// TIA Portal V19 export
FUNCTION_BLOCK "Decoiler_DiameterSensor_FB"   // FB70, LAD
TITLE = COIL DIAMETER ANALOGIC SENSOR MANAGMENT
// stored: MemoryReserve 100, SetENOAutomatically false
   VAR_INPUT
      InLine : Bool;
      AnalogSensor : Int := 0;
      Preset_Conditions : Bool;
      Preset_Button : Bool;
      Preset_Value : Real;
   END_VAR
   VAR_OUTPUT
      CoilDiameter : Real;
   END_VAR
   VAR_IN_OUT
      PersistentValues : Struct
         Data : Struct
            AnalogicSensor_OffsetValue : Real;
            AnalogicSensor_OffsetValid : Bool;
         END_STRUCT;
         Par : Struct
            AnalogicSensor_Enable : Bool;
            AnalogicSensor_RangeLow : Real;
            AnalogicSensor_RangeHigh : Real;
            Diam_Min : Real;
            Diam_Max : Real;
            EndCoil_Diam : Real;
            EndCoil_Timer : Time;
         END_STRUCT;
      END_STRUCT;
      Alarm : Struct
         SensorrPresetNeed : Bool;
      END_STRUCT;
   END_VAR
   VAR
      Sts : Struct
         Standstill : Bool := TRUE;
         AlarmsPresence : Bool;
         WarningsPresence : Bool := FALSE;
         AnalogicSensor_Scale : Real;
         DiameterValueWOOffset : Real;
      END_STRUCT;
      PE_Aux : Bool;
      Filter { S7_SetPoint := 'True'} : "Filter_1°Order";
   END_VAR
   VAR_TEMP
      retval : Word;
      AnalogScaleUnFiletered : Real;
   END_VAR
   VAR_TEMP   // added for the SCL form of the ladder/FBD networks
      _w1 : Bool;
   END_VAR
BEGIN

REGION Network 1: Coil Diameter - Alarm analogic sensor need to be preset
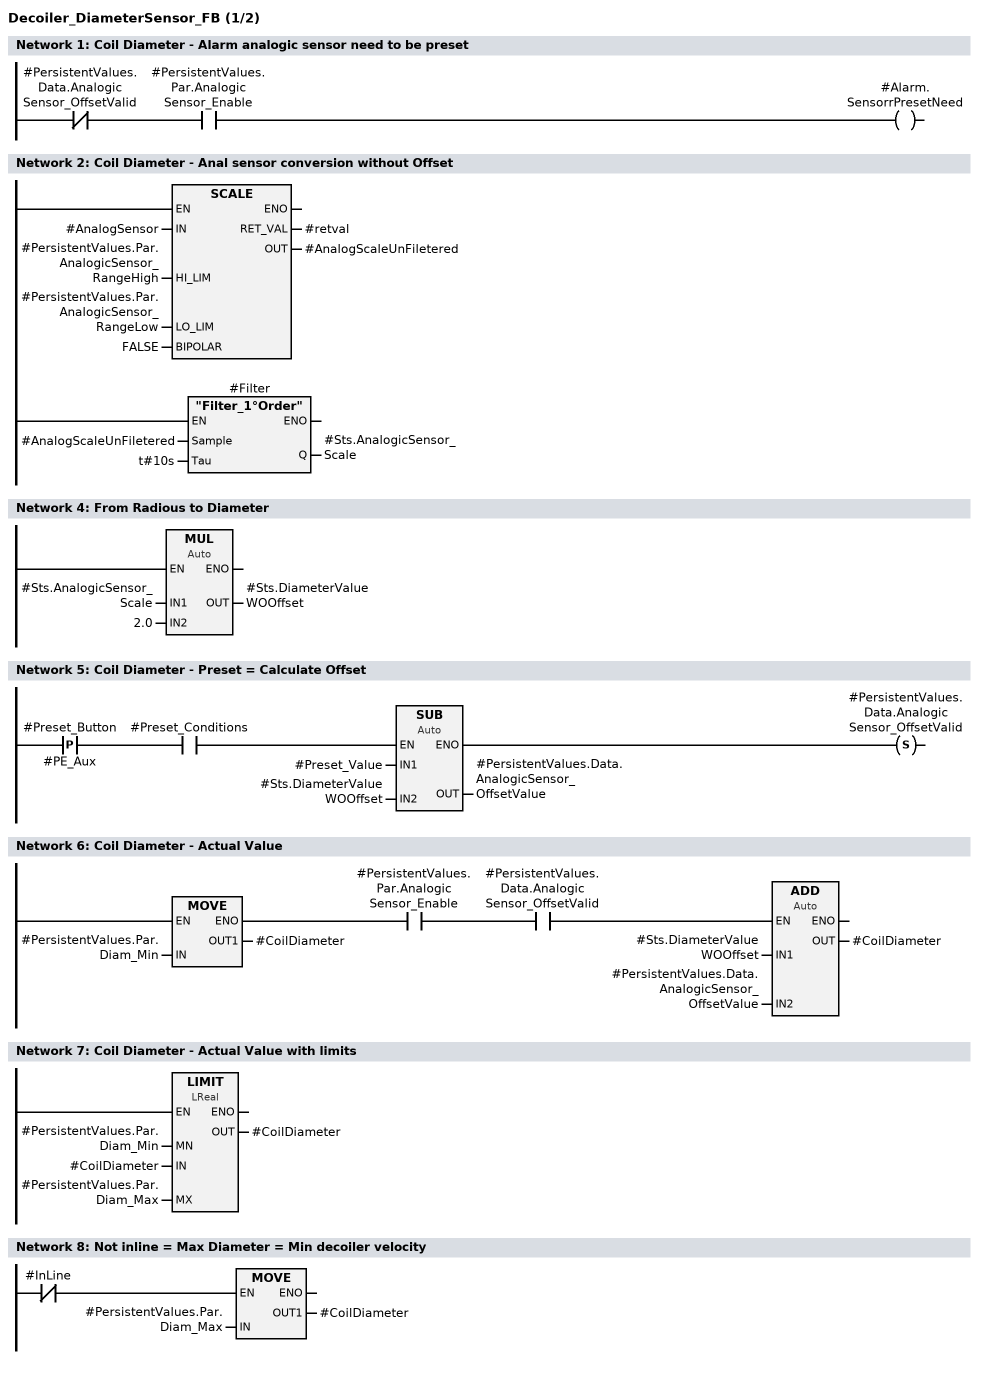
   RUNG wire#powerrail
      I_Contact( #PersistentValues.Data.AnalogicSensor_OffsetValid )
      Contact( #PersistentValues.Par.AnalogicSensor_Enable )
      Coil( #Alarm.SensorrPresetNeed )
   END_RUNG
   // the same network as SCL:
   #Alarm.SensorrPresetNeed := NOT #PersistentValues.Data.AnalogicSensor_OffsetValid AND #PersistentValues.Par.AnalogicSensor_Enable;
END_REGION

REGION Network 2: Coil Diameter - Anal sensor conversion without Offset
   #retval := SCALE(IN := #AnalogSensor,
                    HI_LIM := #PersistentValues.Par.AnalogicSensor_RangeHigh,
                    LO_LIM := #PersistentValues.Par.AnalogicSensor_RangeLow,
                    BIPOLAR := FALSE,
                    OUT => #AnalogScaleUnFiletered);
   #Filter(Sample := #AnalogScaleUnFiletered, Tau := t#10s, Q => #Sts.AnalogicSensor_Scale);   // "Filter_1°Order"
END_REGION

REGION Network 4: From Radious to Diameter
   RUNG wire#powerrail
      { S7_GenerateENO := "TRUE" } Mul(in1 := #Sts.AnalogicSensor_Scale, in2 := 2.0, out => #Sts.DiameterValueWOOffset)
   END_RUNG
   // the same network as SCL:
   #Sts.DiameterValueWOOffset := #Sts.AnalogicSensor_Scale * 2.0;
END_REGION

REGION Network 5: Coil Diameter - Preset = Calculate Offset
   RUNG wire#powerrail
      P_Contact(operand := #Preset_Button, bit := #PE_Aux)
      Contact( #Preset_Conditions )
      Sub(in1 := #Preset_Value, in2 := #Sts.DiameterValueWOOffset, out => #PersistentValues.Data.AnalogicSensor_OffsetValue)
      S_Coil( #PersistentValues.Data.AnalogicSensor_OffsetValid )
   END_RUNG
   // the same network as SCL:
   #_w1 := #Preset_Button AND NOT #PE_Aux;   // rising edge of #Preset_Button
   #PE_Aux := #Preset_Button;
   IF #_w1 AND #Preset_Conditions THEN
       #PersistentValues.Data.AnalogicSensor_OffsetValue := #Preset_Value - #Sts.DiameterValueWOOffset;
       #PersistentValues.Data.AnalogicSensor_OffsetValid := TRUE;
   END_IF;
END_REGION

REGION Network 6: Coil Diameter - Actual Value
   RUNG wire#powerrail
      { S7_GenerateENO := "TRUE" } Move(in := #PersistentValues.Par.Diam_Min, out1 => #CoilDiameter)
      Contact( #PersistentValues.Par.AnalogicSensor_Enable )
      Contact( #PersistentValues.Data.AnalogicSensor_OffsetValid )
      { S7_GenerateENO := "TRUE" } Add(in1 := #Sts.DiameterValueWOOffset, in2 := #PersistentValues.Data.AnalogicSensor_OffsetValue, out => #CoilDiameter)
   END_RUNG
   // the same network as SCL:
   // ENO of a box is taken as its EN; it also drops when the box reports an error
   #CoilDiameter := #PersistentValues.Par.Diam_Min;
   IF #PersistentValues.Par.AnalogicSensor_Enable AND #PersistentValues.Data.AnalogicSensor_OffsetValid THEN
       #CoilDiameter := #Sts.DiameterValueWOOffset + #PersistentValues.Data.AnalogicSensor_OffsetValue;
   END_IF;
END_REGION

REGION Network 7: Coil Diameter - Actual Value with limits
   RUNG wire#powerrail
      { S7_Templates := "value_type := LReal" } Limit(mn := #PersistentValues.Par.Diam_Min, in := #CoilDiameter, mx := #PersistentValues.Par.Diam_Max, out => #CoilDiameter)
   END_RUNG
   // the same network as SCL:
   #CoilDiameter := LIMIT(MN := #PersistentValues.Par.Diam_Min, IN := #CoilDiameter, MX := #PersistentValues.Par.Diam_Max);
END_REGION

REGION Network 8: Not inline = Max Diameter = Min decoiler velocity
   RUNG wire#powerrail
      I_Contact( #InLine )
      { S7_GenerateENO := "TRUE" } Move(in := #PersistentValues.Par.Diam_Max, out1 => #CoilDiameter)
   END_RUNG
   // the same network as SCL:
   IF NOT #InLine THEN #CoilDiameter := #PersistentValues.Par.Diam_Max; END_IF;
END_REGION

REGION Network 9: Alarms presence
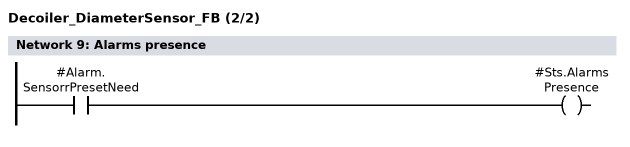
   RUNG wire#powerrail
      Contact( #Alarm.SensorrPresetNeed )
      Coil( #Sts.AlarmsPresence )
   END_RUNG
   // the same network as SCL:
   #Sts.AlarmsPresence := #Alarm.SensorrPresetNeed;
END_REGION
END_FUNCTION_BLOCK
